// TIA Portal V16 export
// export: Created 2020-11-23T18:32:16.2399787Z, ExportSetting WithDefaults, DisplayName Totally Integrated Automation Portal, DisplayVersion V16 Update 2, DisplayName TIA Portal Version Control Interface, DisplayVersion V16 Update 2, DisplayName TIA Portal Openness, DisplayVersion V16 Update 2, DisplayName SINAMICS Startdrive Advanced, DisplayVersion V16 Update 3, DisplayName SINAMICS Startdrive G130, G150, S120, S150, SINAMICS MV, S210, DisplayVersion V16 Update 3, DisplayName SINAMICS Startdrive G110M, G120, G120C, G120D, G120P, G115D, DisplayVersion V16 Update 3, DisplayName STEP 7 Professional, DisplayVersion V16 Update 2, DisplayName STEP 7 Safety, DisplayVersion V16, DisplayName WinCC Professional, DisplayVersion V16 Update 2
FUNCTION_BLOCK "FB1_TESTES"   // FB1, LAD
TITLE = FB para lógicas de testes durante start-up
{ S7_Optimized_Access := 'FALSE' }
AUTHOR : AUT_SIST
NAME : RGrn
VERSION : 0.1
// stored: AutoNumber false, IsIECCheckEnabled false, SetENOAutomatically false, UDAEnableTagReadback false
   VAR DB_SPECIFIC
      TESTE : Bool;
      bit_0_1 : Bool;
      bit_0_2 : Bool;
      bit_0_3 : Bool;
      bit_0_4 : Bool;
      bit_0_5 : Bool;
      bit_0_6 : Bool;
      bit_0_7 : Bool;
      bit_1_0 : Bool;
      bit_1_1 : Bool;
      bit_1_2 : Bool;
      bit_1_3 : Bool;
      bit_1_4 : Bool;
      bit_1_5 : Bool;
      bit_1_6 : Bool;
      bit_1_7 : Bool;
      eBosch_FO1_InCy : Bool;
      eBosch_FO1_CyCmp : Bool;
      eBosch_Ch0_1_OK : Bool;
      eBosch_Ch0_2_OK : Bool;
      eBosch_Ch0_3_OK : Bool;
      eBosch_Ch1_1_OK : Bool;
      eBosch_Ch1_2_OK : Bool;
      eBosch_Ch1_3_OK : Bool;
      eBosch_FO2_InCy : Bool;
      eBosch_FO2_CyCmp : Bool;
      eBosch_Ch2_1_OK : Bool;
      eBosch_Ch2_2_OK : Bool;
      eBosch_Ch2_3_OK : Bool;
      eBosch_Ch2_4_OK : Bool;
      bit_3_6 : Bool;
      bit_3_7 : Bool;
      bit_4_0 : Bool;
      bit_4_1 : Bool;
      bit_4_2 : Bool;
      bit_4_3 : Bool;
      bit_4_4 : Bool;
      bit_4_5 : Bool;
      bit_4_6 : Bool;
      bit_4_7 : Bool;
      FP_0 : Bool;
      FP_1 : Bool;
      FP_2 : Bool;
      FP_3 : Bool;
      FP_4 : Bool;
      FP_5 : Bool;
      FP_6 : Bool;
      FP_7 : Bool;
   END_VAR
   VAR_TEMP
      RET_VAL_FC455 : Word;
      Aux_Soma_rodas : Real;
      Med_Rot_rodas : Real;
      Med_parcial_rel_trm : Real;
      Retval_SFC20 : Int;   // Auxiliar armazenamento de mensagens do SFC20
      zero : DWord;
   END_VAR
BEGIN
END_FUNCTION_BLOCK
